Staubli VAL3: onInsert.pgx

public program onInsert(string& x_sItem[])
  local string l_sEvent
begin
  cls()
  call selectType(l_sEvent)
  // exit
  if l_sEvent==""
    x_sItem=""
    return
  endIf
  //
  if x_sItem!="IF"
    // compose the instruction
    call make_NUM(l_sEvent)
  else
    // usine an IF
    call make_if(l_sEvent)
  endIf
  // update
  x_sItem=l_sEvent
end
